  PROC DrawPart37()
    MoveL Offs(pOrigin,39.61,104.48,0.00),v60,z0,tPen\WObj:=wPaper;
    MoveL Offs(pOrigin,39.61,97.28,0.00),v40,z0,tPen\WObj:=wPaper;
    MoveL Offs(pOrigin,40.66,97.57,0.00),v40,z0,tPen\WObj:=wPaper;
    MoveL Offs(pOrigin,40.66,106.58,0.00),v40,fine,tPen\WObj:=wPaper;
    MoveL Offs(pOrigin,40.66,106.58,6.00),v60,z5,tPen\WObj:=wPaper;
    MoveL Offs(pOrigin,45.94,108.38,6.00),vTravel,z5,tPen\WObj:=wPaper;
    MoveL Offs(pOrigin,45.94,108.38,0.00),v60,z0,tPen\WObj:=wPaper;
    MoveL Offs(pOrigin,45.94,122.47,0.00),v40,fine,tPen\WObj:=wPaper;
    MoveL Offs(pOrigin,45.94,122.47,6.00),v60,z5,tPen\WObj:=wPaper;
    MoveL Offs(pOrigin,47.00,123.37,6.00),vTravel,z5,tPen\WObj:=wPaper;
    MoveL Offs(pOrigin,47.00,123.37,0.00),v60,z0,tPen\WObj:=wPaper;
    MoveL Offs(pOrigin,47.00,109.72,0.00),v40,fine,tPen\WObj:=wPaper;
    MoveL Offs(pOrigin,47.00,109.72,6.00),v60,z5,tPen\WObj:=wPaper;
    MoveL Offs(pOrigin,37.50,100.57,6.00),vTravel,z5,tPen\WObj:=wPaper;
    MoveL Offs(pOrigin,37.50,100.57,0.00),v60,z0,tPen\WObj:=wPaper;
    MoveL Offs(pOrigin,37.50,96.22,0.00),v40,fine,tPen\WObj:=wPaper;
    MoveL Offs(pOrigin,37.50,96.22,6.00),v60,z5,tPen\WObj:=wPaper;
    MoveL Offs(pOrigin,51.95,89.62,6.00),vTravel,z5,tPen\WObj:=wPaper;
    MoveL Offs(pOrigin,51.95,89.62,0.00),v60,z0,tPen\WObj:=wPaper;
    MoveL Offs(pOrigin,53.30,89.62,0.00),v40,fine,tPen\WObj:=wPaper;
    MoveL Offs(pOrigin,53.30,89.62,6.00),v60,z5,tPen\WObj:=wPaper;
    MoveL Offs(pOrigin,48.06,129.22,6.00),vTravel,z5,tPen\WObj:=wPaper;
    MoveL Offs(pOrigin,48.06,129.22,0.00),v60,z0,tPen\WObj:=wPaper;
    MoveL Offs(pOrigin,48.06,131.17,0.00),v40,z0,tPen\WObj:=wPaper;
    MoveL Offs(pOrigin,49.11,131.32,0.00),v40,z0,tPen\WObj:=wPaper;
    MoveL Offs(pOrigin,49.11,130.12,0.00),v40,fine,tPen\WObj:=wPaper;
    MoveL Offs(pOrigin,49.11,130.12,6.00),v60,z5,tPen\WObj:=wPaper;
  ENDPROC

ENDMODULE
